FUNCTION_BLOCK FB_JobInfoPublisher IMPLEMENTS I_JobInfo, I_Observable
VAR CONSTANT
	MAX_OBSERVERS : UDINT := 5;
END_VAR
VAR_INPUT
END_VAR
VAR_OUTPUT
END_VAR
VAR
	_observers		: ARRAY [1..MAX_OBSERVERS] OF I_Observer;
	_title	  		: T_MaxString;	// Subject text of event
	_last_state 	: E_FutureExecutionState; // Job state before transition.
	_new_state 		: E_FutureExecutionState; // Job state after transition.
	_record_time	: T_FILETIME64; // File-time at the time of transition.
	_job			: I_Job; // Reference to job instance of which transition occurs.
	_error_id		: HRESULT;
END_VAR

METHOD add_observer : BOOL
VAR_INPUT
	observer	: I_Observer;
END_VAR
VAR
	i : UDINT;
END_VAR
FOR i := 1 TO MAX_OBSERVERS DO
	IF _observers[i] = 0 THEN
		_observers[i] := observer;
		_error_id := S_OK;
		add_observer := TRUE;
		RETURN;
	END_IF
END_FOR
_error_id := -1;
add_observer := TRUE;
END_METHOD

PROPERTY error_id : HRESULT
GET
error_id := _error_id;
END_GET
SET
_error_id := error_id;
END_SET
END_PROPERTY

PROPERTY job : I_Job
GET
job := _job;
END_GET
SET
_job := job;
END_SET
END_PROPERTY

{warning 'Add property implementation'}
PROPERTY last_state : E_FutureExecutionState
GET
last_state := _last_state;
END_GET
SET
_last_state := last_state;
END_SET
END_PROPERTY

{warning 'Add property implementation'}
PROPERTY new_state : E_FutureExecutionState
GET
new_state := _new_state;
END_GET
SET
_new_state := new_state;
END_SET
END_PROPERTY

METHOD notify_observers : BOOL
VAR
	i : UDINT;
END_VAR
notify_observers := TRUE;
FOR i := 1 TO MAX_OBSERVERS DO
	IF _observers[i] <> 0 THEN
		_observers[i].notify(THIS^);
	END_IF
END_FOR
END_METHOD

PROPERTY record_time : T_FILETIME64
GET
record_time := _record_time;
END_GET
SET
_record_time := record_time;
END_SET
END_PROPERTY

METHOD remove_observer : BOOL
VAR_INPUT
	observer	: I_Observer;
END_VAR
VAR
	i : UDINT;
END_VAR
FOR i := 1 TO MAX_OBSERVERS DO
	IF _observers[i] = observer THEN
		_observers[i] := 0;
		_error_id := S_OK;
		remove_observer := TRUE;
		RETURN;
	END_IF
END_FOR
_error_id := -2;
remove_observer := TRUE;
END_METHOD

{warning 'Add property implementation'}
PROPERTY title : T_MaxString
GET
title := _title;
END_GET
SET
_title := title;
END_SET
END_PROPERTY

END_FUNCTION_BLOCK

(* stored: Version 1.1.0.1, ProductVersion 3.1.4026.13
   POU FB_JobInfoPublisher: Id {7a64fcb3-a887-456a-9fd8-a111e49a6cf3}, SpecialFunc None
   Method add_observer: Id {d712393b-074b-40ce-ab34-a3ae158e8435}
   Property error_id: Id {097bfdb5-8c91-4f30-951c-7994a4445464}
   Get Get: Id {c8873fe5-6f71-431e-be62-a1683a1d1ef5}
   Set Set: Id {77d00a62-3027-4c5d-bf1e-5e6680cf3218}
   Property job: Id {7ffe74ad-75ab-4ffd-be67-8bd95da67896}
   Get Get: Id {203eace5-176a-4546-9ba8-9222c3581386}
   Set Set: Id {3d8f4474-bc71-4648-8e41-4fee6b02a08d}
   Property last_state: Id {04fd2377-5fcc-4370-8438-cd220270ddf8}
   Get Get: Id {a4a76b6e-bad7-4637-9b1e-10d9cd0435c0}
   Set Set: Id {786bc1c9-24e5-4fd2-bfbd-3220e2794ff2}
   Property new_state: Id {0f0d0773-d759-4533-b954-ab8abc3edd0b}
   Get Get: Id {67ebf388-b35b-48e6-9a2a-3a5df0b4c462}
   Set Set: Id {915ab9e3-bd11-4fc8-b718-cdd764d0a9e3}
   Method notify_observers: Id {24198e8b-93da-4bfe-b178-70a0f1f8b69b}
   Property record_time: Id {e043bb70-f943-4c44-93c4-10e25e34e9f8}
   Get Get: Id {1ef59afb-5415-4e15-ad52-c1f7e22fbdec}
   Set Set: Id {eda5ceb4-28bd-460e-b13d-925e46216f1b}
   Method remove_observer: Id {ee66de95-751f-40b3-aa1d-da1581a9b056}
   Property title: Id {df3f22e1-8fa7-4ede-9800-4f7f70c43c3a}
   Get Get: Id {57c6140d-176b-4ab3-b731-538428ec1e7e}
   Set Set: Id {e471fcef-a8fd-4f1d-a8b2-0a5063e37ba2} *)
